// TIA Portal V20 export
DATA_BLOCK "DB_RX"   // DB13
{ S7_Optimized_Access := 'FALSE' }
   VAR
      Lifebit : Bool;
      Start_Curing : Bool;
      open_door_1 : Bool;
      close_door_1 : Bool;
      open_door_2 : Bool;
      close_door_2 : Bool;
      open_door_3 : Bool;
      close_door_3 : Bool;
      Setpoint_Temperature : Int;
      Setpoint_Humidity : Int;
      Reserve_byte : Byte;
   END_VAR
BEGIN
END_DATA_BLOCK
